FUNCTION_BLOCK dvSensor
VAR_INPUT
END_VAR
VAR_OUTPUT
END_VAR
VAR
	ModeActual		: E_GEMMA := E_GEMMA.A6Inicializando;
	Name			: STRING; 				// Nombre del actuador, p.ej. K_1
	prValue			: BOOL := FALSE;		// Valor previo para detectar cambios de estado	
	hwValue AT %I*	: BOOL;					// Vinculación al hardware de la estación
	uiValue			: BOOL;					// Vinculación a la visualización
	uiToolTip		: STRING;				// Tooltip en la visualización
	uiEnabled		: BOOL := FALSE; 		// Deshabilitar el control cuando hay conexión con el hardware
END_VAR

METHOD ProcessCycle : BOOL
VAR_INPUT
	ModeActual	: E_GEMMA := E_GEMMA.A6Inicializando;
END_VAR

VAR_OUTPUT
	sfcValue 	: BOOL;		// estado del sensor que se entregará al Grafcet
END_VAR
uiEnabled := TRUE; // (ModeActual = E_GEMMA.F4VerificacionSinOrden); // Planta habilitado sólo en modo F4
 
IF uiEnabled THEN
	// Si está ejecutando en local, simular que el hardware a recibido el valor de la visualización
	hwValue := uiValue;	
ELSE
	hwValue := sfcValue;
	uiValue := sfcValue;
END_IF
sfcValue := uiValue;		// estado del sensor que se entregará al Grafcet
END_METHOD

END_FUNCTION_BLOCK

(* stored: Version 1.1.0.1, ProductVersion 3.1.4024.11
   POU dvSensor: Id {c4029391-ebd0-4ae7-8ab5-3338cf1cc185}, SpecialFunc None
   Method ProcessCycle: Id {71ee41d9-0d14-4d00-a8c7-99dc223f0a9d} *)
